FUNCTION_BLOCK CLIENT_2 (* Two-Item Client Interface *)
  (* Standard: 61499-2 *)
  (* Version 0.0, 2004-10-21, JHC, Rockwell Automation, Converted from SRC version. *)
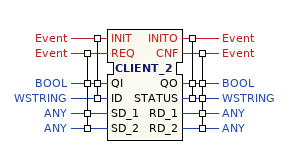
  EVENT_INPUT
    INIT WITH QI, ID; (* Service Initialization *)
    REQ WITH QI, SD_1, SD_2; (* Service Request *)
  END_EVENT
  EVENT_OUTPUT
    INITO WITH QO, STATUS; (* Initialization Confirm *)
    CNF WITH QO, STATUS, RD_1, RD_2; (* Service Confirmation *)
  END_EVENT
  VAR_INPUT
    QI : BOOL; (* Event Input Qualifier *)
    ID : WSTRING; (* Connection Identifier *)
    SD_1 : ANY; (* Data to Send *)
    SD_2 : ANY; (* Data to Send *)
  END_VAR
  VAR_OUTPUT
    QO : BOOL; (* Event Output Qualifier *)
    STATUS : WSTRING; (* Service Status *)
    RD_1 : ANY; (* Received Data *)
    RD_2 : ANY; (* Received Data *)
  END_VAR
END_FUNCTION_BLOCK
